(* PLC project Unnamed, Unknown Unnamed 1 *)
(* stored: creationDateTime 2025-05-23T23:38:38, modificationDateTime 2025-05-23T23:57:20 *)

PROGRAM ConveyorStarter
  VAR
    visionSensor AT %IX0.0 : BOOL;
    exitSensor AT %IX0.2 : BOOL;
    converyorMotor AT %QX0.6 : BOOL;
  END_VAR

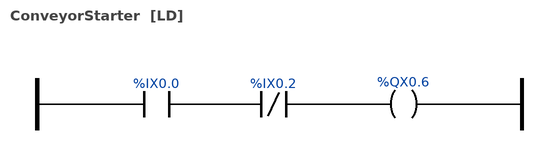
(* LD diagram, written out as Structured Text *)
%QX0.6 := %IX0.0 AND NOT %IX0.2;
END_PROGRAM

CONFIGURATION Config0
  RESOURCE Res0 ON PLC
    TASK task0(INTERVAL := T#20ms, PRIORITY := 0);
    PROGRAM instance0 WITH task0 : ConveyorStarter;
  END_RESOURCE
END_CONFIGURATION
